// TIA Portal V18 export
DATA_BLOCK "ST10_SysOutput"   // DB1002
{ S7_Optimized_Access := 'TRUE' }
// stored: AutoNumber false, MemoryReserve 100
   VAR
      oTowerLight : Struct
         Red : Bool;
         Yellow : Bool;
         Green : Bool;
         Blue : Bool;
      END_STRUCT;
      HMIButtonLight : Struct
         ControlOn : Bool := false;   // HMI_上电按钮
         ControlOff : Bool;   // HMI_断电按钮
         MachineStart : Bool := false;   // HMI_设备启动按钮
         MachineStop : Bool := false;   // HMI_设备停止按钮
         ResetButton : Bool := false;   // HMI_复位按钮
         "Manual/Auto" : Bool := false;   // HMI_手/自动切换按钮
         SafetyGateUnlock : Bool := false;   // HMI_安全门解锁按钮
      END_STRUCT;
      BoxLight : Struct
         oMachineStartLight : Bool;   // 启动按钮PB
         oMachineStopLight : Bool;   // 停止按钮PB
         oResetLight : Bool;   // 复位按钮PB
         oSafetyGateUnlockLight : Bool;   // 安全门解锁按钮PB
      END_STRUCT;
      SafetyDoorCoil : Array[1..20] of Bool;
      MaterialDoorCoil : Array[1..20] of Bool;
   END_VAR
BEGIN
END_DATA_BLOCK
